// TIA Portal V16 export
// export: Created 2021-07-12T14:47:20.9180027Z, ExportSetting WithDefaults, DisplayName Totally Integrated Automation Portal, DisplayVersion V16, DisplayName TIA Portal Version Control Interface, DisplayVersion V16, DisplayName TIA Portal Openness, DisplayVersion V16, DisplayName STEP 7 Professional, DisplayVersion V16, DisplayName STEP 7 Safety, DisplayVersion V16, DisplayName WinCC Professional, DisplayVersion V16
TYPE "SimaHydTO_typeHMIConnectionVCharEditorStatus"
TITLE = SimaHydTO_typeHMIConnectionVCharEditorStatus
// HMI interface: VChar editor - Status (PLC -> HMI)
// stored: IsFailsafeCompliant false
   STRUCT
      EditorActive : Bool;
      SaveAsSelected : Bool;
      Busy : Bool;
      Error : Bool;
      VCharLoad { S7_SetPoint := 'True'} : "SimaHydTO_typeHMIConnectionVCharSelectorStatus";
      VCharSave { S7_SetPoint := 'True'} : "SimaHydTO_typeHMIConnectionVCharSelectorStatus";
   END_STRUCT;
END_TYPE
